TYPE FlexChain :
STRUCT
	pdo AT %I* : ARRAY[0..31] OF BYTE;//max pdo inputs of the flex chain bus
END_STRUCT
END_TYPE

(* stored: Version 1.1.0.1, ProductVersion 3.1.4024.15
   DUT FlexChain: Id {48b81f7d-6f62-4c8f-b5ef-72489a412e55} *)
